PROGRAM main
VAR_INPUT
	X0 : bool;
	X1 : bool;
	X2 : bool;
END_VAR

VAR_OUTPUT
	Y0 : bool;
	Y1 : bool;
	Y2 : bool;
END_VAR

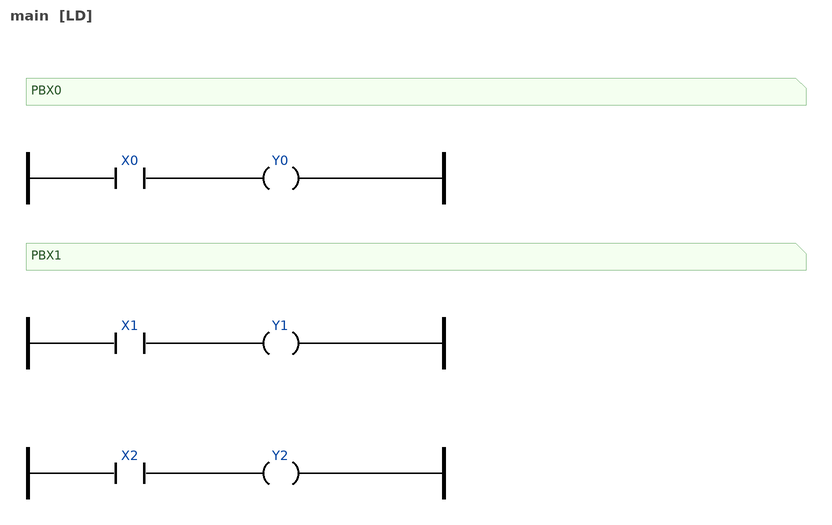
(* LD diagram, written out as Structured Text *)
(* PBX0 *)
Y0 := X0;
(* PBX1 *)
Y1 := X1;
Y2 := X2;
END_PROGRAM
